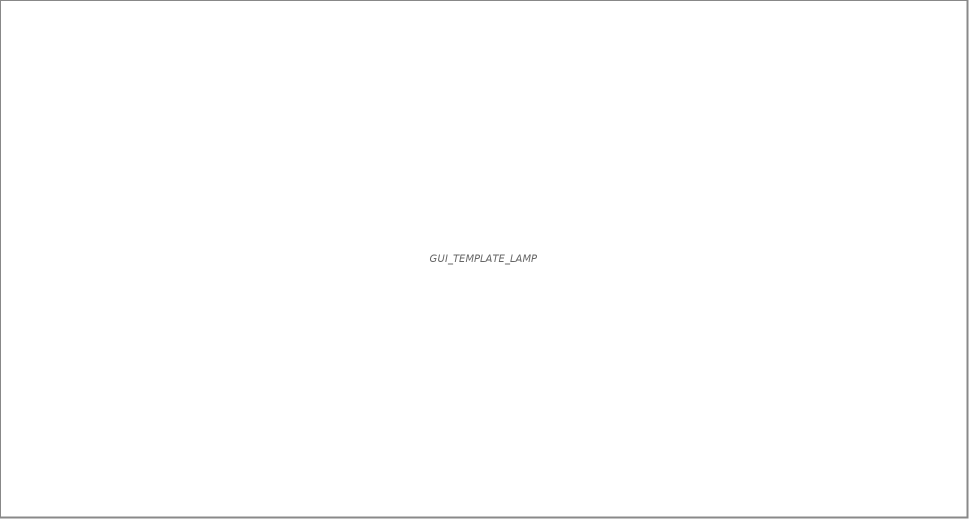
VISUALIZATION GUI_Lamp001  // 969x519
    Frame (0,0 967x517)
        shows GUI_TEMPLATE_LAMP(m_Instance := MAIN.Lamp001)
END_VISUALIZATION

(* stored: Version 1.1.0.1, ProductVersion 3.1.4024.3
   Visu GUI_Lamp001: Id {ba6b4829-cfe8-4c1b-80a7-d8c3b6d4dc60} *)
